{attribute 'hide_all_locals'}
FUNCTION_BLOCK FB_Symo_PV_Inverter_FLOAT_1_DM_1_Inverter
VAR_INPUT PERSISTENT
	bEnable						: BOOL;												//True = Function is enabled, FALSE = Function is dissabled, no new Data
	sIPAdress					: STRING(15);										//IP Adress from the Inverter
	byUnitID_Inverter			: BYTE;												//Unit ID fromt the Inverter (1 to 247)
END_VAR
VAR_OUTPUT
	stDataSymo10				: ST_Symo_PV_OutData;								//Output structure with Data from Symo 10
	stDataEMPower_PV			: ST_ElectricMeter_Output_Power;					//Output structure with Data from Electric Meter PV (Power Data)
	stDataEMCounter_PV			: ST_ElectricMeter_Output_Counter;					//Output structure with Data from Electric Meter PV (Counter Data)
	diNrOfEM_OUT_PV				: DINT;												//Active Number from the Electric Meter for using on other functions
END_VAR
VAR
	fbElMeter					: FB_ElectricMeter;									//Electric Meter Function 
	fbNumberDevice				: FB_NumberOfDevice;								//Function block to calcualte the number of the Device
	fbConvertEnergyRegister		: FB_CV_WORD_TO_DWORD;								//Convert function
	fbMBRead_FC3				: FB_MBReadRegs;									//Modbus Read Function (FC3)
	timDelay					: TON;												//Timer for Delay between Requests
	timTimeout					: TON;												//Timer for Timeout
	timDissableFunctions		: TON;												//Timer to dissable the Function after Lynus_Standards.Constants_General.tTimeDissableLynusFunctions Days without connection to the Lynus Cloud
	timResetConnectionOnGVL		: TON;												//Timer to try reset the connection Flag on the GVL. (When somebody delete the Connection Function and make only a onlinechange)
	FPEnable					: R_TRIG;											//Internal positive Edge
	FPError_FC_3				: R_TRIG;											//Internal positive Edge
	PD_String					: FB_PersistentData_String;							//Function to save persistent data 
	stFloat						: ST_UN_FLOAT_CONVERT_DWORD_REAL;					//Convert the Float Raw Value
	arrBuffer_FC3				: ARRAY[1..47] OF WORD;								//Buffer with Data from FC3
	arrPD						: ARRAY[1..2] OF FB_PersistentData_Number;			//Function to save persistent data 
	byWaitInStep				: BYTE;												//Wait in Step before start to clean data on PLC
	iStateGVLData				: INT;												//State machine to handle the data on the GVL
	iStateModbus				: INT;												//State variable for Statemachine
	iStateModbus_CP				: INT;												//Compare State variable
	diCounterForGVL				: DINT;												//Counter to clean old data on GVL
	lrCheckValue				: LREAL;											//Internal Value to check the value before convert
END_VAR

//Creator : Kai Ebensperger
//Company : Lynus AG
//Date : 28.04.2021
//Version : 1.0.0.0

//With this function its possible to read out values from the Symo 10 PV Inverter from the factory Fronius
//This Function read out the Values from 1 Fronius Datamanager with maximal 1 Inverter.
//The protocol to the Inverter is Modbus TCP
//Versions that are supported : 1.1.5-0
//Attention. To access the registers, an offset of 1 must always be subtracted. Register 40001 would then be on register 40000.
//This Function use the FLOAT Format

//NOTE for diNr.....Designation => 
//_IN = Here Data come in from other Functions or go out to other functions about the GVL
//_OUT = Here Data go out to other functions about the GVL

(*------------------------------------------------------------------------------------------General Input Part---------------------------------------------------------------------------------------------*)

//Check limitation
byUnitID_Inverter := LIMIT(1,byUnitID_Inverter,247);

(*-------------------------------------------------------------Calcualte the number of EM System---------------------------------------------------------------*)

fbNumberDevice(
	diActualNumberOfDevices:= Lynus_Standards.GVL_Energy.stNumberOfDevices.diNumberOfElectricMeters, 
	diMaxNumberOfDevices:= Constants_Energy.diMaxNumberOfElectricMeters, 
	udiCounterOnlineChange:= TwinCAT_SystemInfoVarList._AppInfo.OnlineChangeCnt, 
	bNumberIsCalculatet=> , 
	bFPNumberIsCalculatet=> , 
	bOnlineChange=> , 
	diNumberForThisDevice=> diNrOfEM_OUT_PV, 
	diNumberOfTotalDevices=> );

//Write new Numer on GVL
IF fbNumberDevice.bFPNumberIsCalculatet THEN
	Lynus_Standards.GVL_Energy.stNumberOfDevices.diNumberOfElectricMeters := fbNumberDevice.diNumberOfTotalDevices;	
END_IF 

//Delete old Number on GVL
IF fbNumberDevice.bOnlineChange THEN 
	Lynus_Standards.GVL_Energy.stNumberOfDevices.diNumberOfElectricMeters := diNrOfEM_OUT_PV;	
		iStateGVLData := 1; 
END_IF

(*-------------------------------------------------------------Service from Backend is ready and check the connection to backen for dissabel/enable Function---------------------------------------------------------------*)

//Try to reset the variable for connection on the GVL. When all is normal then the Lynus Mqtt connection function set this variable to true in the next cycle
//When we have no connection to the backend then after Lynus_Standards.Constants_General.tTimeDissableLynusFunctions days the Function is dissabled with all of his functionalities
timResetConnectionOnGVL(IN:= NOT timResetConnectionOnGVL.Q, PT:= T#1H, Q=> , ET=> );
	IF timResetConnectionOnGVL.Q THEN Lynus_Standards.GVL_Communicator.bStateConnectionToEnableFunctions := FALSE; END_IF
		IF NOT Lynus_Standards.GVL_Communicator.bStateConnectionToEnableFunctions THEN timDissableFunctions.IN := TRUE; ELSE timDissableFunctions.IN := FALSE; END_IF  
			timDissableFunctions(IN:= , PT:= Lynus_Standards.Constants_General.tTimeDissableLynusFunctions, Q=> , ET=> );
	
(*------------------------------------------------------------------------------------------State Machine---------------------------------------------------------------------------------------------*)
	
//Enable
FPEnable(CLK:= bEnable, Q=> );
	IF FPEnable.Q AND iStateModbus = 0 THEN iStateModbus := 1; END_IF
		IF NOT bEnable OR timDissableFunctions.Q THEN iStateModbus := 0; END_IF

//Timer for delay
timDelay(IN:= , PT:= T#100MS, Q=> , ET=> );	

//Timer for Timeout in Statemachine
	IF iStateModbus = iStateModbus_CP THEN timTimeout.IN := TRUE; ELSE timTimeout.IN := FALSE; END_IF
		IF iStateModbus = 0 THEN timTimeout.IN := FALSE; END_IF
timTimeout(IN:= , PT:= T#20S, Q=> , ET=> );	

//Statemachine
CASE iStateModbus OF
	
	0://Init Step
		iStateModbus_CP := iStateModbus;
			timDelay.IN := FALSE;
		
		stDataSymo10.bFunctionIsActive := FALSE;
			stDataSymo10.eOperatingStateInverter := E_Symo_PV_OperatingState.eNoDataReceived;
				fbMBRead_FC3.bExecute := FALSE;
					lrCheckValue := 0;
									
	1://Read out first Registers from 40072 to 40118
		stDataSymo10.bFunctionIsActive := TRUE;
			iStateModbus_CP := iStateModbus;
		
		fbMBRead_FC3.nQuantity := 47;
			fbMBRead_FC3.nMBAddr := 40071;
				fbMBRead_FC3.bExecute := TRUE;
					fbMBRead_FC3.nUnitID := byUnitID_Inverter;
			
		IF fbMBRead_FC3.bBusy THEN timDelay.IN := TRUE; END_IF
		
		//Wait for Delay, copy Data and then next step
		IF NOT fbMBRead_FC3.bBusy AND NOT fbMBRead_FC3.bError AND timDelay.Q THEN
			//Copy Data Current L1
			fbConvertEnergyRegister(wInputValue_1:= arrBuffer_FC3[3], wInputValue_2:= arrBuffer_FC3[4], eByteOrderForConvert:= eByteOrder.eBigEndian, dwOutputValue=> );
				stFloat.dwRawValue := fbConvertEnergyRegister.dwOutputValue;
					lrCheckValue := stFloat.rValueFloat;	
						IF lrCheckValue >= - 3.402823E+38 AND lrCheckValue <= 3.402823E+38 THEN 
							fbElMeter.lrCurrentL1 := lrCheckValue;
						ELSE
							iStateModbus := 300;
								stDataSymo10.eErrorState := E_Symo_PV_Error.eSymo10TooBigValueReceived;		
						END_IF
			//Copy Data Current L2
			fbConvertEnergyRegister(wInputValue_1:= arrBuffer_FC3[5], wInputValue_2:= arrBuffer_FC3[6], eByteOrderForConvert:= eByteOrder.eBigEndian, dwOutputValue=> );
				stFloat.dwRawValue := fbConvertEnergyRegister.dwOutputValue;
					lrCheckValue := stFloat.rValueFloat;	
						IF lrCheckValue >= - 3.402823E+38 AND lrCheckValue <= 3.402823E+38 THEN 
							fbElMeter.lrCurrentL2 := lrCheckValue;
						ELSE
							iStateModbus := 300;
								stDataSymo10.eErrorState := E_Symo_PV_Error.eSymo10TooBigValueReceived;		
						END_IF
			//Copy Data Current L3
			fbConvertEnergyRegister(wInputValue_1:= arrBuffer_FC3[7], wInputValue_2:= arrBuffer_FC3[8], eByteOrderForConvert:= eByteOrder.eBigEndian, dwOutputValue=> );
				stFloat.dwRawValue := fbConvertEnergyRegister.dwOutputValue;
					lrCheckValue := stFloat.rValueFloat;	
						IF lrCheckValue >= - 3.402823E+38 AND lrCheckValue <= 3.402823E+38 THEN 
							fbElMeter.lrCurrentL3 := lrCheckValue;
						ELSE
							iStateModbus := 300;
								stDataSymo10.eErrorState := E_Symo_PV_Error.eSymo10TooBigValueReceived;		
						END_IF
			//Copy Data Voltage L1-L2
			fbConvertEnergyRegister(wInputValue_1:= arrBuffer_FC3[9], wInputValue_2:= arrBuffer_FC3[10], eByteOrderForConvert:= eByteOrder.eBigEndian, dwOutputValue=> );
				stFloat.dwRawValue := fbConvertEnergyRegister.dwOutputValue;
					lrCheckValue := stFloat.rValueFloat;	
						IF lrCheckValue >= - 3.402823E+38 AND lrCheckValue <= 3.402823E+38 THEN 
							fbElMeter.lrVoltageL1L2 := lrCheckValue;
						ELSE
							iStateModbus := 300;
								stDataSymo10.eErrorState := E_Symo_PV_Error.eSymo10TooBigValueReceived;		
						END_IF
			//Copy Data Voltage L2-L3
			fbConvertEnergyRegister(wInputValue_1:= arrBuffer_FC3[11], wInputValue_2:= arrBuffer_FC3[12], eByteOrderForConvert:= eByteOrder.eBigEndian, dwOutputValue=> );
				stFloat.dwRawValue := fbConvertEnergyRegister.dwOutputValue;
					lrCheckValue := stFloat.rValueFloat;	
						IF lrCheckValue >= - 3.402823E+38 AND lrCheckValue <= 3.402823E+38 THEN 
							fbElMeter.lrVoltageL2L3 := lrCheckValue;
						ELSE
							iStateModbus := 300;
								stDataSymo10.eErrorState := E_Symo_PV_Error.eSymo10TooBigValueReceived;		
						END_IF
			//Copy Data Voltage L3-L1
			fbConvertEnergyRegister(wInputValue_1:= arrBuffer_FC3[13], wInputValue_2:= arrBuffer_FC3[14], eByteOrderForConvert:= eByteOrder.eBigEndian, dwOutputValue=> );
				stFloat.dwRawValue := fbConvertEnergyRegister.dwOutputValue;
					lrCheckValue := stFloat.rValueFloat;	
						IF lrCheckValue >= - 3.402823E+38 AND lrCheckValue <= 3.402823E+38 THEN 
							fbElMeter.lrVoltageL3L1 := lrCheckValue;
						ELSE
							iStateModbus := 300;
								stDataSymo10.eErrorState := E_Symo_PV_Error.eSymo10TooBigValueReceived;		
						END_IF
			//Copy Data Voltage L1-N
			fbConvertEnergyRegister(wInputValue_1:= arrBuffer_FC3[15], wInputValue_2:= arrBuffer_FC3[16], eByteOrderForConvert:= eByteOrder.eBigEndian, dwOutputValue=> );
				stFloat.dwRawValue := fbConvertEnergyRegister.dwOutputValue;
					lrCheckValue := stFloat.rValueFloat;	
						IF lrCheckValue >= - 3.402823E+38 AND lrCheckValue <= 3.402823E+38 THEN 
							fbElMeter.lrVoltageL1N := lrCheckValue;
						ELSE
							iStateModbus := 300;
								stDataSymo10.eErrorState := E_Symo_PV_Error.eSymo10TooBigValueReceived;		
						END_IF
			//Copy Data Voltage L2-N
			fbConvertEnergyRegister(wInputValue_1:= arrBuffer_FC3[17], wInputValue_2:= arrBuffer_FC3[18], eByteOrderForConvert:= eByteOrder.eBigEndian, dwOutputValue=> );
				stFloat.dwRawValue := fbConvertEnergyRegister.dwOutputValue;
					lrCheckValue := stFloat.rValueFloat;	
						IF lrCheckValue >= - 3.402823E+38 AND lrCheckValue <= 3.402823E+38 THEN 
							fbElMeter.lrVoltageL2N := lrCheckValue;
						ELSE
							iStateModbus := 300;
								stDataSymo10.eErrorState := E_Symo_PV_Error.eSymo10TooBigValueReceived;		
						END_IF
			//Copy Data Voltage L3-N
			fbConvertEnergyRegister(wInputValue_1:= arrBuffer_FC3[19], wInputValue_2:= arrBuffer_FC3[20], eByteOrderForConvert:= eByteOrder.eBigEndian, dwOutputValue=> );
				stFloat.dwRawValue := fbConvertEnergyRegister.dwOutputValue;
					lrCheckValue := stFloat.rValueFloat;	
						IF lrCheckValue >= - 3.402823E+38 AND lrCheckValue <= 3.402823E+38 THEN 
							fbElMeter.lrVoltageL3N := lrCheckValue;
						ELSE
							iStateModbus := 300;
								stDataSymo10.eErrorState := E_Symo_PV_Error.eSymo10TooBigValueReceived;		
						END_IF
			//Copy Data AC Power
			fbConvertEnergyRegister(wInputValue_1:= arrBuffer_FC3[21], wInputValue_2:= arrBuffer_FC3[22], eByteOrderForConvert:= eByteOrder.eBigEndian, dwOutputValue=> );
				stFloat.dwRawValue := fbConvertEnergyRegister.dwOutputValue;
					lrCheckValue := stFloat.rValueFloat;	
						IF lrCheckValue >= - 3.402823E+38 AND lrCheckValue <= 3.402823E+38 THEN 
							fbElMeter.lrPowerTotal := lrCheckValue;
						ELSE
							iStateModbus := 300;
								stDataSymo10.eErrorState := E_Symo_PV_Error.eSymo10TooBigValueReceived;		
						END_IF
			//Copy Data Frequency
			fbConvertEnergyRegister(wInputValue_1:= arrBuffer_FC3[23], wInputValue_2:= arrBuffer_FC3[24], eByteOrderForConvert:= eByteOrder.eBigEndian, dwOutputValue=> );
				stFloat.dwRawValue := fbConvertEnergyRegister.dwOutputValue;
					lrCheckValue := stFloat.rValueFloat;	
						IF lrCheckValue >= - 3.402823E+38 AND lrCheckValue <= 3.402823E+38 THEN 
							fbElMeter.lrFrequency := lrCheckValue;
						ELSE
							iStateModbus := 300;
								stDataSymo10.eErrorState := E_Symo_PV_Error.eSymo10TooBigValueReceived;		
						END_IF
			//Copy Data Apparent Power
			fbConvertEnergyRegister(wInputValue_1:= arrBuffer_FC3[25], wInputValue_2:= arrBuffer_FC3[26], eByteOrderForConvert:= eByteOrder.eBigEndian, dwOutputValue=> );
				stFloat.dwRawValue := fbConvertEnergyRegister.dwOutputValue;
					lrCheckValue := stFloat.rValueFloat;	
						IF lrCheckValue >= - 3.402823E+38 AND lrCheckValue <= 3.402823E+38 THEN 
							fbElMeter.lrApparentPowerTotal := lrCheckValue;
						ELSE
							iStateModbus := 300;
								stDataSymo10.eErrorState := E_Symo_PV_Error.eSymo10TooBigValueReceived;		
						END_IF
			//Copy Data Reactive Power
			fbConvertEnergyRegister(wInputValue_1:= arrBuffer_FC3[27], wInputValue_2:= arrBuffer_FC3[28], eByteOrderForConvert:= eByteOrder.eBigEndian, dwOutputValue=> );
				stFloat.dwRawValue := fbConvertEnergyRegister.dwOutputValue;
					lrCheckValue := stFloat.rValueFloat;	
						IF lrCheckValue >= - 3.402823E+38 AND lrCheckValue <= 3.402823E+38 THEN 
							fbElMeter.lrReactivePowerTotal := lrCheckValue;
						ELSE
							iStateModbus := 300;
								stDataSymo10.eErrorState := E_Symo_PV_Error.eSymo10TooBigValueReceived;		
						END_IF
			//Copy Data AC production Energy
			fbConvertEnergyRegister(wInputValue_1:= arrBuffer_FC3[31], wInputValue_2:= arrBuffer_FC3[32], eByteOrderForConvert:= eByteOrder.eBigEndian, dwOutputValue=> );
				stFloat.dwRawValue := fbConvertEnergyRegister.dwOutputValue;
					lrCheckValue := stFloat.rValueFloat;	
						IF lrCheckValue >= - 3.402823E+38 AND lrCheckValue <= 3.402823E+38 THEN 
							fbElMeter.lrCounterEnergyT1_Production := lrCheckValue / 1000;
								fbElMeter.lrTotalCounterEnergy_Production := fbElMeter.lrCounterEnergyT1_Production;
						ELSE
							iStateModbus := 300;
								stDataSymo10.eErrorState := E_Symo_PV_Error.eSymo10TooBigValueReceived;		
						END_IF
			//Operating State		
			IF arrBuffer_FC3[47] = 1 THEN stDataSymo10.eOperatingStateInverter := E_Symo_PV_OperatingState.eOff;
				ELSIF arrBuffer_FC3[47] = 2 THEN stDataSymo10.eOperatingStateInverter := E_Symo_PV_OperatingState.eSleeping;
				ELSIF arrBuffer_FC3[47] = 3 THEN stDataSymo10.eOperatingStateInverter := E_Symo_PV_OperatingState.eStartingUp;
				ELSIF arrBuffer_FC3[47] = 4 THEN stDataSymo10.eOperatingStateInverter := E_Symo_PV_OperatingState.eTrackingPowerPoint;
				ELSIF arrBuffer_FC3[47] = 5 THEN stDataSymo10.eOperatingStateInverter := E_Symo_PV_OperatingState.eForcedPowerReduction;
				ELSIF arrBuffer_FC3[47] = 6 THEN stDataSymo10.eOperatingStateInverter := E_Symo_PV_OperatingState.eShuttingDown;
				ELSIF arrBuffer_FC3[47] = 7 THEN stDataSymo10.eOperatingStateInverter := E_Symo_PV_OperatingState.eFaults;
				ELSIF arrBuffer_FC3[47] = 8 THEN stDataSymo10.eOperatingStateInverter := E_Symo_PV_OperatingState.eStandby;
				ELSE stDataSymo10.eOperatingStateInverter := E_Symo_PV_OperatingState.eNoDataReceived;
			END_IF
			//Next Step
			IF iStateModbus = 1 THEN
				fbMBRead_FC3.bExecute := FALSE;
					timDelay.IN := FALSE;
						iStateModbus := 2;
							stDataSymo10.bError := FALSE; 
								stDataSymo10.eErrorState := E_Symo_PV_Error.eNoError;
			END_IF
		END_IF
			
		//Error from Inverter
		IF NOT fbMBRead_FC3.bBusy AND NOT fbMBRead_FC3.bError AND timDelay.Q AND stDataSymo10.eOperatingStateInverter = E_Symo_PV_OperatingState.eFaults THEN
			iStateModbus := 300;
				stDataSymo10.eErrorState := E_Symo_PV_Error.eSymo10Error;
		END_IF
	 
		//Error or Timeout
		IF FPError_FC_3.Q OR timTimeout.Q THEN
			iStateModbus := 300;
				stDataSymo10.eErrorState := E_Symo_PV_Error.eModbusTCPError;
		END_IF

	2://Wait and back to 1 step
		iStateModbus_CP := iStateModbus;
		
			iStateModbus := 1;
				
	300://Error
		iStateModbus_CP := iStateModbus;
			timDelay.IN := FALSE;
				fbMBRead_FC3.bExecute := FALSE;
					stDataSymo10.bError := TRUE;
						iStateModbus := 1;				
							
END_CASE

(*------------------------------------------------------------------------------------------Modbus TCP Function---------------------------------------------------------------------------------------------*)

fbMBRead_FC3(sIPAddr:= sIPAdress, nTCPPort:= 502, cbLength:= SIZEOF(arrBuffer_FC3), pDestAddr:= ADR(arrBuffer_FC3), tTimeout:= T#10S );
	FPError_FC_3(CLK:= fbMBRead_FC3.bError, Q=> );

(*----------------------------------------------------------------------------------------Electric Meter Data----------------------------------------------------------------------------------------------*)

//Error and Warning
IF timDissableFunctions.Q THEN fbElMeter.bWarning := TRUE; fbElMeter.iWarningCode := 0; ELSE fbElMeter.bWarning := FALSE; END_IF   
	IF stDataSymo10.bError OR Lynus_Standards.GVL_Energy.stNumberOfDevices.diNumberOfElectricMeters > Constants_Energy.diMaxNumberOfElectricMeters THEN fbElMeter.bError := TRUE; ELSE fbElMeter.bError := FALSE; END_IF  

IF Lynus_Standards.GVL_Energy.stNumberOfDevices.diNumberOfElectricMeters > Constants_Energy.diMaxNumberOfElectricMeters THEN fbElMeter.iErrorCode := 1;
ELSIF stDataSymo10.bError THEN fbElMeter.iErrorCode := 0;
END_IF  

//Read Out Data done for EM Function
IF iStateModbus <> 2 THEN fbElMeter.bReadOutDataDone := TRUE; ELSE fbElMeter.bReadOutDataDone := FALSE; END_IF

//Function block for meter data
fbElMeter(
	bEnable:= bEnable AND NOT timDissableFunctions.Q, 
	bError:= , 
	bEnableReadOutFunction:= FALSE, 
	bWriteWithDelay:= TRUE,
	bPowerDataInvers:= TRUE, 
	bReadOutDataDone:= ,
	iTimeReadOutInterval:= , 
	iErrorCode:= , 
	iWarningCode:= , 
	lrTotalCounterEnergy_Consumption:= 0, 
	lrTotalCounterEnergy_Production:= , 
	lrCounterEnergyT1_Consumption:= 0, 
	lrCounterEnergyT2_Consumption:= 0, 
	lrCounterEnergyT1_Production:= , 
	lrCounterEnergyT2_Production:= 0, 
	lrCurrentL1:= , 
	lrVoltageL1N:= , 
	lrVoltageL1L2:= , 
	lrPowerL1:= 0, 
	lrCurrentL2:= , 
	lrVoltageL2N:= , 
	lrVoltageL2L3:= , 
	lrPowerL2:= 0, 
	lrCurrentL3:= , 
	lrVoltageL3N:= , 
	lrVoltageL3L1:= , 
	lrPowerL3:= 0, 
	lrPowerTotal:= , 
	lrFrequency:= , 
	lrReactivePowerTotal:= , 
	lrApparentPowerTotal:= , 
	tTimDelayOutput:= T#5S, 
	stDataEMOutPower=> , 
	stDataEMOutPowerDelay=> stDataEMPower_PV, 
	stDataEMOutCounter=> ,
	stDataEMOutCounterDelay=> stDataEMCounter_PV, 
	bReadOutMeter=> );

(*-----------------------------------------------------------Handle data to Global structure for the Electric Meter system-----------------------------------------------------------------*)

CASE iStateGVLData OF
	
	0://Init Step
		byWaitInStep := 0;
			diCounterForGVL := 1;
	
	1://Wait for 4 Steps before clean al Data on GVL
		byWaitInStep := byWaitInStep + 1;
			IF byWaitInStep >= 4 AND fbNumberDevice.bNumberIsCalculatet THEN iStateGVLData := 2; END_IF
				//To much Devices, back to the Init step
				IF byWaitInStep >= 4 AND NOT fbNumberDevice.bNumberIsCalculatet THEN iStateGVLData := 0; END_IF	
			
	2://Clear all Data in GVL
		Lynus_Standards.GVL_Energy.stDataElectricMeters[diCounterForGVL].bEnabled := FALSE;	
			Lynus_Standards.GVL_Energy.stDataElectricMeters[diCounterForGVL].byErrorWarning := 0;
				Lynus_Standards.GVL_Energy.stDataElectricMeters[diCounterForGVL].lrCounterEnergyT1_Consumption := 0;
					Lynus_Standards.GVL_Energy.stDataElectricMeters[diCounterForGVL].lrCounterEnergyT1_Production := 0;
						Lynus_Standards.GVL_Energy.stDataElectricMeters[diCounterForGVL].lrCounterEnergyT2_Consumption := 0;
							Lynus_Standards.GVL_Energy.stDataElectricMeters[diCounterForGVL].lrCounterEnergyT2_Production := 0;
								Lynus_Standards.GVL_Energy.stDataElectricMeters[diCounterForGVL].lrPower := 0;
									Lynus_Standards.GVL_Energy.stDataElectricMeters[diCounterForGVL].lrPowerConsumption := 0;
										Lynus_Standards.GVL_Energy.stDataElectricMeters[diCounterForGVL].lrPowerConsumption := 0;
											Lynus_Standards.GVL_Energy.stDataElectricMeters[diCounterForGVL].lrPowerProduction := 0;
												Lynus_Standards.GVL_Energy.stDataElectricMeters[diCounterForGVL].lrTotalCounterEnergy_Consumption := 0;
													Lynus_Standards.GVL_Energy.stDataElectricMeters[diCounterForGVL].lrTotalCounterEnergy_Production := 0;
		
		diCounterForGVL := diCounterForGVL + 1;
			diCounterForGVL := LIMIT(0,diCounterForGVL,Constants_Energy.diMaxNumberOfElectricMeters);
				//Back to the init step
				IF diCounterForGVL >= Constants_Energy.diMaxNumberOfElectricMeters THEN iStateGVLData := 0; END_IF

END_CASE 	 

IF diNrOfEM_OUT_PV > 0 AND fbNumberDevice.bNumberIsCalculatet THEN
	Lynus_Standards.GVL_Energy.stDataElectricMeters[diNrOfEM_OUT_PV].bEnabled := fbElMeter.stDataEMOutPower.bEnabled;
		Lynus_Standards.GVL_Energy.stDataElectricMeters[diNrOfEM_OUT_PV].byErrorWarning := fbElMeter.stDataEMOutPower.byErrorWarning;
			Lynus_Standards.GVL_Energy.stDataElectricMeters[diNrOfEM_OUT_PV].lrCounterEnergyT1_Consumption := fbElMeter.stDataEMOutCounter.lrCounterEnergyT1_Consumption;
				Lynus_Standards.GVL_Energy.stDataElectricMeters[diNrOfEM_OUT_PV].lrCounterEnergyT1_Production := fbElMeter.stDataEMOutCounter.lrCounterEnergyT1_Production;
					Lynus_Standards.GVL_Energy.stDataElectricMeters[diNrOfEM_OUT_PV].lrCounterEnergyT2_Consumption := fbElMeter.stDataEMOutCounter.lrCounterEnergyT2_Consumption;
						Lynus_Standards.GVL_Energy.stDataElectricMeters[diNrOfEM_OUT_PV].lrCounterEnergyT2_Production := fbElMeter.stDataEMOutCounter.lrCounterEnergyT2_Production;		
							Lynus_Standards.GVL_Energy.stDataElectricMeters[diNrOfEM_OUT_PV].lrPower := fbElMeter.stDataEMOutPower.lrPowerTotal;
								Lynus_Standards.GVL_Energy.stDataElectricMeters[diNrOfEM_OUT_PV].lrPowerConsumption := fbElMeter.stDataEMOutPower.lrPowerConsumption;
									Lynus_Standards.GVL_Energy.stDataElectricMeters[diNrOfEM_OUT_PV].lrPowerProduction := fbElMeter.stDataEMOutPower.lrPowerProduction;
										Lynus_Standards.GVL_Energy.stDataElectricMeters[diNrOfEM_OUT_PV].lrTotalCounterEnergy_Consumption := fbElMeter.stDataEMOutCounter.lrTotalCounterEnergy_Consumption;
											Lynus_Standards.GVL_Energy.stDataElectricMeters[diNrOfEM_OUT_PV].lrTotalCounterEnergy_Production := fbElMeter.stDataEMOutCounter.lrTotalCounterEnergy_Production;
END_IF

(*----------------------------------------------------------Save persistent data----------------------------------------------------------------*)

arrPD[1](lrValue:= BOOL_TO_LREAL(bEnable), bEventBasedActive=> );
arrPD[2](lrValue:= BYTE_TO_LREAL(byUnitID_Inverter), bEventBasedActive=> );
PD_String(sText:= sIPAdress, bEventBasedActive=> );

END_FUNCTION_BLOCK

(* stored: Version 1.1.0.1, ProductVersion 3.1.4024.9
   POU FB_Symo_PV_Inverter_FLOAT_1_DM_1_Inverter: Id {0d2c64c6-6860-4373-b5e0-b35de35065ea}, SpecialFunc None *)
